FUNCTION_BLOCK WagoSystemWithIOWithNetworking (* Composite Function Block Type *)
  (* Standard: 61499-2 *)
  (* Version 0.2, 2003-12-05, JHC, Rockwell Automation, Renamed from NEWCOMPFB. *)
  (* Compiler header: package fb.rt.wago; *)
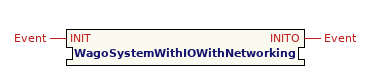
  EVENT_INPUT
    INIT; (* Initialization Request *)
  END_EVENT
  EVENT_OUTPUT
    INITO; (* Initialization Confirm *)
  END_EVENT
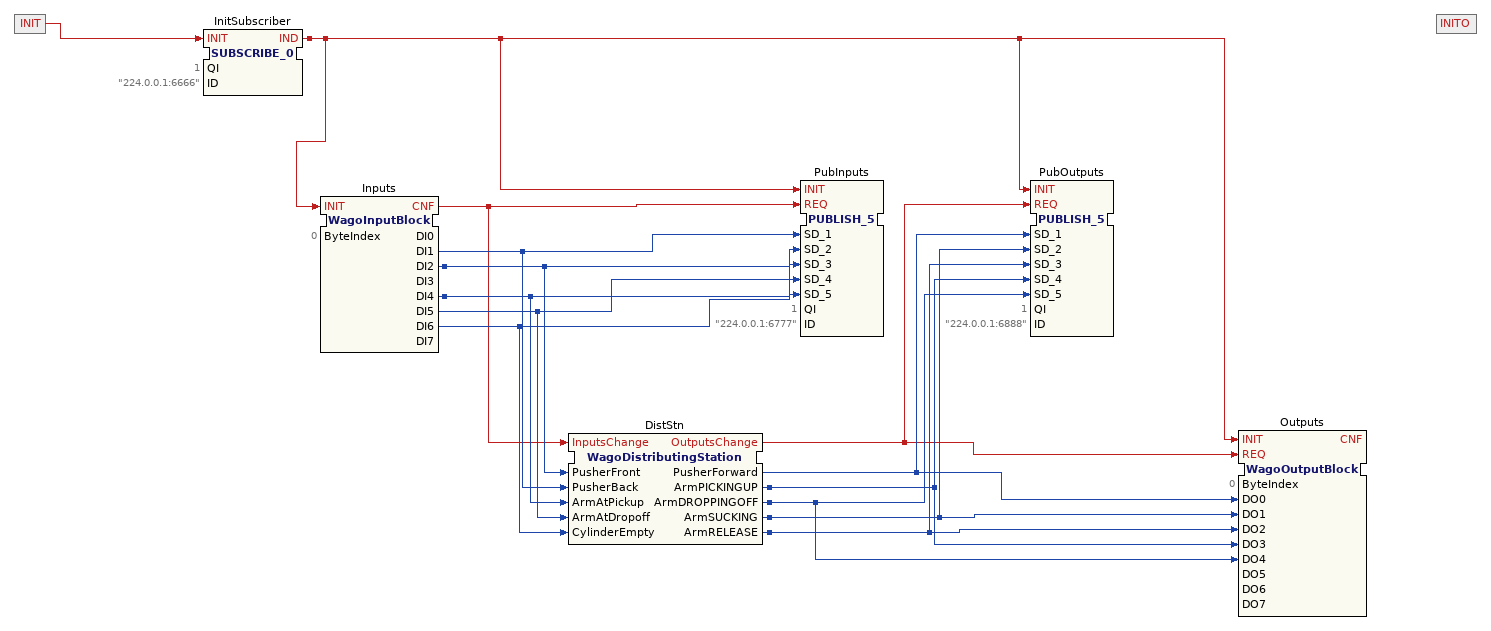
  FBS
    DistStn : WagoDistributingStation;
    Inputs : WagoInputBlock(ByteIndex := 0);
    Outputs : WagoOutputBlock(ByteIndex := 0);
    PubInputs : PUBLISH_5(QI := 1, ID := "224.0.0.1:6777");
    PubOutputs : PUBLISH_5(QI := 1, ID := "224.0.0.1:6888");
    InitSubscriber : SUBSCRIBE_0(QI := 1, ID := "224.0.0.1:6666");
  END_FBS
  EVENT_CONNECTIONS
    INIT TO InitSubscriber.INIT;
    InitSubscriber.IND TO Inputs.INIT;
    InitSubscriber.IND TO PubInputs.INIT;
    InitSubscriber.IND TO PubOutputs.INIT;
    InitSubscriber.IND TO Outputs.INIT;
    Inputs.CNF TO DistStn.InputsChange;
    DistStn.OutputsChange TO Outputs.REQ;
    Inputs.CNF TO PubInputs.REQ;
    DistStn.OutputsChange TO PubOutputs.REQ;
  END_CONNECTIONS
  DATA_CONNECTIONS
    Inputs.DI2 TO DistStn.PusherFront;
    Inputs.DI1 TO DistStn.PusherBack;
    Inputs.DI4 TO DistStn.ArmAtPickup;
    Inputs.DI5 TO DistStn.ArmAtDropoff;
    Inputs.DI6 TO DistStn.CylinderEmpty;
    DistStn.PusherForward TO Outputs.DO0;
    DistStn.ArmPICKINGUP TO Outputs.DO3;
    DistStn.ArmDROPPINGOFF TO Outputs.DO4;
    DistStn.ArmSUCKING TO Outputs.DO1;
    DistStn.ArmRELEASE TO Outputs.DO2;
    Inputs.DI1 TO PubInputs.SD_1;
    Inputs.DI2 TO PubInputs.SD_2;
    Inputs.DI4 TO PubInputs.SD_3;
    Inputs.DI5 TO PubInputs.SD_4;
    Inputs.DI6 TO PubInputs.SD_5;
    DistStn.PusherForward TO PubOutputs.SD_1;
    DistStn.ArmSUCKING TO PubOutputs.SD_2;
    DistStn.ArmRELEASE TO PubOutputs.SD_3;
    DistStn.ArmPICKINGUP TO PubOutputs.SD_4;
    DistStn.ArmDROPPINGOFF TO PubOutputs.SD_5;
  END_CONNECTIONS
END_FUNCTION_BLOCK
